TYPE "MEStoPLC_MainCheckInStation1ST350_ext"
VERSION : 0.1
   STRUCT
      PartTypeID : Int;
      Station1PalletID : Int;
      Station1PartSN : String[60];
      DataMatrixPartSN : String[60];
      Spare : Array[128..199] of Byte;
      Massage { S7_SetPoint := 'False'} : "MEStoPLC_AlarmMassage_ext";
   END_STRUCT;

END_TYPE

